Staubli VAL3: start.pgx

program start()
begin
  do
    for i=0 to 4
      movej(a[i],flange,vit)
    endFor
    movej(s,flange,vitesse)
    movel(w,flange,vitesse)
    waitEndMove()
  until (false)
end
